// TwinCAT 3 PLC project Untitled1
// ProgramVersion: 3.1.4024.0
// libraries:
//   SPT Base Types, * (Beckhoff Automation LLC)
//   SPT Utilities, * (Beckhoff Automation LLC)
//   Tc2_Standard, * (Beckhoff Automation GmbH)
//   Tc2_System, * (Beckhoff Automation GmbH)
//   Tc3_Module, * (Beckhoff Automation GmbH)
//   Tc3_PackML_V2, * (Beckhoff Automation GmbH)
// project tree:
//   DUTs/ E_EquipmentModuleList.TcDUT
//   Interfaces/ ITF_Observable.TcIO, ITF_Observer.TcIO
//   / PlcTask.TcTTO
//   POUs/ CD_Observer.TcCD (not stored), EquipmentModule.TcPOU, Interlock.TcPOU, MachineModule.TcPOU, MAIN.TcPOU
// real-time tasks:
//   TASK PlcTask: cycle T#10ms, priority 20, ADS port 350

CONFIGURATION Untitled1
    RESOURCE PLC ON TwinCAT3
        TASK PlcTask(INTERVAL := T#10ms, PRIORITY := 20);
        PROGRAM MAIN WITH PlcTask : MAIN;
    END_RESOURCE
END_CONFIGURATION

// ---- DUTs/E_EquipmentModuleList.TcDUT
{attribute 'qualified_only'}
{attribute 'strict'}
{attribute 'to_string'}
TYPE E_EquipmentModuleList :
(
	Open := 0,//Interlock is open and available
	EM1,
	EM2,
	EM3,
	Last
);
END_TYPE

// ---- Interfaces/ITF_Observable.TcIO
INTERFACE ITF_Observable

METHOD notifyObserverConnection : BOOL
END_METHOD

METHOD registerObserver : BOOL
VAR_INPUT
	Observer : ITF_Observer;
END_VAR
END_METHOD

METHOD removeObserver : BOOL
VAR_INPUT
	Observer : ITF_Observer;
END_VAR
END_METHOD

END_INTERFACE

// ---- Interfaces/ITF_Observer.TcIO
INTERFACE ITF_Observer

METHOD updateConnection
VAR_INPUT
	Module : REFERENCE TO MachineModule;
END_VAR
END_METHOD

METHOD updateLock
VAR_INPUT
	setLock : BOOL;
END_VAR
END_METHOD

END_INTERFACE

// ---- POUs/MAIN.TcPOU
PROGRAM MAIN
VAR
	Machine : MachineModule := (Name := 'Machine');	
END_VAR

Machine.CyclicLogic();

END_PROGRAM

// ---- POUs/MachineModule.TcPOU
FUNCTION_BLOCK MachineModule EXTENDS FB_PackML_BaseModule IMPLEMENTS ITF_Observable
VAR
	//SubModules
	Equip1 : EquipmentModule := (Name := 'EM1');
	Equip2 : EquipmentModule := (Name := 'EM2');
	Equip3 : EquipmentModule := (Name := 'EM3');

	//ITF_Observable
	_Observers : ARRAY[1..Parameters_PackML_Base.MAX_NO_OF_SUBMODULES + 1] OF ITF_Observer;

	//Data to be Observered
	_InterlockList	  : E_EquipmentModuleList;
	interlockListPrev : E_EquipmentModuleList;

	//CyclicLogic
	fbRT	  : R_TRIG;
	register1 : BOOL;
	remove1	  : BOOL;
	register2 : BOOL;
	remove2	  : BOOL;
	register3 : BOOL;
	remove3	  : BOOL;
END_VAR

METHOD PUBLIC CyclicLogic
IF NOT _InitComplete THEN
	_InitComplete := Initialize();
	RETURN;
END_IF

//On data change call all observers
fbRT(CLK := _InterlockList <> interlockListPrev);
IF fbRT.Q THEN
	IF _InterlockList = E_EquipmentModuleList.Open THEN
		notifyObserverLock(setLock := FALSE);
	ELSE
		notifyObserverLock(setLock := TRUE);
	END_IF

	interlockListPrev := _InterlockList;
END_IF

//Attach Observer
IF register1 THEN
	IF registerObserver(Equip1) THEN
		register1 := FALSE;
	END_IF
END_IF

IF register2 THEN
	IF registerObserver(Equip2) THEN
		register2 := FALSE;
	END_IF
END_IF

IF register3 THEN
	IF registerObserver(Equip3) THEN
		register3 := FALSE;
	END_IF
END_IF

//Detach Observer
IF remove1 THEN
	IF removeObserver(Equip1) THEN
		Unlock(Equip1);
		remove1 := FALSE;
	END_IF
END_IF

IF remove2 THEN
	IF removeObserver(Equip2) THEN
		Unlock(Equip2);
		remove2 := FALSE;
	END_IF
END_IF

IF remove3 THEN
	IF removeObserver(Equip3) THEN
		Unlock(Equip3);
		remove3 := FALSE;
	END_IF
END_IF

SUPER^.CyclicLogic();
END_METHOD

METHOD PROTECTED Initialize : BOOL
Initialize := FALSE;
CASE DescendantSequenceState OF
	0:
		//
		RegisterSubmodule(Equip1);
		RegisterSubmodule(Equip2);
		RegisterSubmodule(Equip3);

		//
		registerObserver(Equip1);
		registerObserver(Equip2);
		registerObserver(Equip3);

		//
		_LogModeChanges			:= FALSE;
		_LogStateChanges		:= FALSE;
		DescendantSequenceState := DescendantSequenceState + 10;

	10:
		(* Call the Super *)
		IF SUPER^.Initialize() THEN
			DescendantSequenceState := DescendantSequenceState + 10;
		END_IF

	20:
		Initialize := TRUE;
END_CASE
END_METHOD

PROPERTY InterlockList : E_EquipmentModuleList
GET
InterlockList := _InterlockList;
END_GET
END_PROPERTY

METHOD PUBLIC Lock : BOOL
VAR_INPUT
	EM : REFERENCE TO FB_PackML_BaseModule;
END_VAR

VAR
	eList : E_EquipmentModuleList;
END_VAR
//Select the element from the ENUM that matches a string value
FOR eList := E_EquipmentModuleList.Open TO E_EquipmentModuleList.Last DO
	IF EM.Name = TO_STRING(eList) THEN
		_InterlockList := eList;//Set the enum instance to the element that holds the lock
		EXIT;
	END_IF
END_FOR
END_METHOD

METHOD notifyObserverConnection : BOOL
VAR
	i : udint;
END_VAR
//Call all registered Observers and pass them the Observable
FOR i := 1 TO Parameters_PackML_Base.MAX_NO_OF_SUBMODULES DO
	IF _Observers[i] <> 0 THEN
		_Observers[i].updateConnection(THIS^);
	END_IF
END_FOR
END_METHOD

METHOD notifyObserverLock : BOOL
VAR_INPUT
	setLock : BOOL;
END_VAR
VAR
	i: UDINT;
END_VAR
//Call all registered Observers and pass them the lock value
FOR i := 1 TO Parameters_PackML_Base.MAX_NO_OF_SUBMODULES DO
	IF _Observers[i] <> 0 THEN
		_Observers[i].updateLock(setLock);
	END_IF
END_FOR
END_METHOD

METHOD registerObserver : BOOL
VAR_INPUT
	Observer : ITF_Observer;
END_VAR

VAR
	i : UDINT;
END_VAR
registerObserver := FALSE;

//Check if Observer is already registered
FOR i := 1 TO Parameters_PackML_Base.MAX_NO_OF_SUBMODULES DO
	IF _Observers[i] = Observer THEN
		RETURN;
	END_IF
END_FOR

//Add Observer to first available index within the array
FOR i := 1 TO Parameters_PackML_Base.MAX_NO_OF_SUBMODULES DO
	IF _Observers[i] = 0 THEN
		_Observers[i] := Observer;
		_Observers[i].updateConnection(THIS^); //On registration pass Observable to Observer for any Initialization it might need to do
		registerObserver := TRUE;
		EXIT;
	END_IF
END_FOR
END_METHOD

METHOD removeObserver : BOOL
VAR_INPUT
	Observer : ITF_Observer;
END_VAR

VAR
	i : UDINT;
END_VAR
removeObserver := FALSE;

//Check for valid input
IF (Observer = 0) THEN
	RETURN;
END_IF

//Find Observer to be removed and set the array index to 0
FOR i := 1 TO Parameters_PackML_Base.MAX_NO_OF_SUBMODULES DO
	IF (_Observers[i] = Observer) THEN
		Observer.updateLock(setLock := FALSE);
		Observer.updateConnection(0);//Let the Observer know that it no longer has an Observable
		_Observers[i]  := 0;
		removeObserver := TRUE;
		EXIT;
	END_IF
END_FOR

//Clean up array
FOR i := 1 TO Parameters_PackML_Base.MAX_NO_OF_SUBMODULES DO
	IF _Observers[i] = 0 THEN
		//array size is declared to +1 for these 2 lines of code to be safe
		_Observers[i]	  := _Observers[i + 1];
		_Observers[i + 1] := 0;
	END_IF
END_FOR
END_METHOD

METHOD Unlock : bool
VAR_INPUT
	EM : REFERENCE TO FB_PackML_BaseModule;
END_VAR
VAR
	eList : E_EquipmentModuleList;
END_VAR
//If the EM that called the method is holding the lock, then remove the lock
FOR eList := E_EquipmentModuleList.Open TO E_EquipmentModuleList.Last DO
	IF EM.Name = TO_STRING(_InterlockList) THEN
		_InterlockList := E_EquipmentModuleList.Open;
		EXIT;
	END_IF
END_FOR
END_METHOD

END_FUNCTION_BLOCK

// ---- POUs/EquipmentModule.TcPOU
FUNCTION_BLOCK EquipmentModule EXTENDS FB_PackML_BaseModule IMPLEMENTS ITF_Observer
VAR
	NextState		: BOOL;
	AbortReq		: BOOL;
	
	
	//ITF_Observable
	OModule : REFERENCE TO MachineModule;

	//
	interlock : Interlock;
	reqDoStuff: BOOL;
	stuffDone: BOOL;
END_VAR

METHOD PUBLIC CyclicLogic
VAR
END_VAR
IF NOT _InitComplete THEN
	_InitComplete := Initialize();
	RETURN;
END_IF

//Check Interlock
IF reqDoStuff THEN
	reqDoStuff := FALSE;
	IF interlock.Unlocked THEN
		IF __ISVALIDREF(OModule) THEN
			OModule.Lock(THIS^); //Lock the interlock
		END_IF

		//OK to do stuff
	ELSE
		//Locked
		IF __ISVALIDREF(OModule) THEN
			TRACE(CONCAT(STR1 := 'Interlock set by: ', STR2 := TO_STRING(OModule.InterlockList)));
		END_IF
	END_IF
END_IF

//Release Interlock
IF stuffDone AND interlock.Locked THEN
	stuffDone := FALSE;
	IF __ISVALIDREF(OModule) THEN
		OModule.Unlock(THIS^);
	END_IF
END_IF

SUPER^.CyclicLogic();
END_METHOD

METHOD PROTECTED Initialize : BOOL
Initialize := TRUE;
END_METHOD

METHOD updateConnection
VAR_INPUT
	Module : REFERENCE TO MachineModule;
END_VAR
OModule REF= Module;
END_METHOD

METHOD updateLock
VAR_INPUT
	setLock : BOOL;
END_VAR
//Method called by observable to notify of lock status
IF setLock THEN
	interlock.Lock();
ELSE
	interlock.Unlock();
END_IF
END_METHOD

END_FUNCTION_BLOCK

// ---- POUs/Interlock.TcPOU
FUNCTION_BLOCK Interlock
VAR
	_Locked : BOOL;
END_VAR

METHOD Lock : BOOL
VAR_INPUT
END_VAR
_Locked := TRUE;
END_METHOD

PROPERTY Locked : bool
GET
Locked := _Locked;
END_GET
END_PROPERTY

METHOD Unlock : BOOL
VAR_INPUT
END_VAR
_Locked := false;
END_METHOD

PROPERTY Unlocked : bool
GET
Unlocked := NOT _Locked;
END_GET
END_PROPERTY

END_FUNCTION_BLOCK
